PROGRAM PRG_Test
VAR
	tableSerializerTest : TableSerializerTest;
END_VAR

TcUnit.RUN();

END_PROGRAM

(* stored: Version 1.1.0.1, ProductVersion 3.1.4024.12
   POU PRG_Test: Id {68af6fdb-1ffc-4105-a501-ed469ea4d0b7}, SpecialFunc None *)
